// Mitsubishi GX Works2 project: Q03udv LG   PLC: Q03UDV
// ZONE 6 MOD 2021 06072021

PROGRAM MAIN
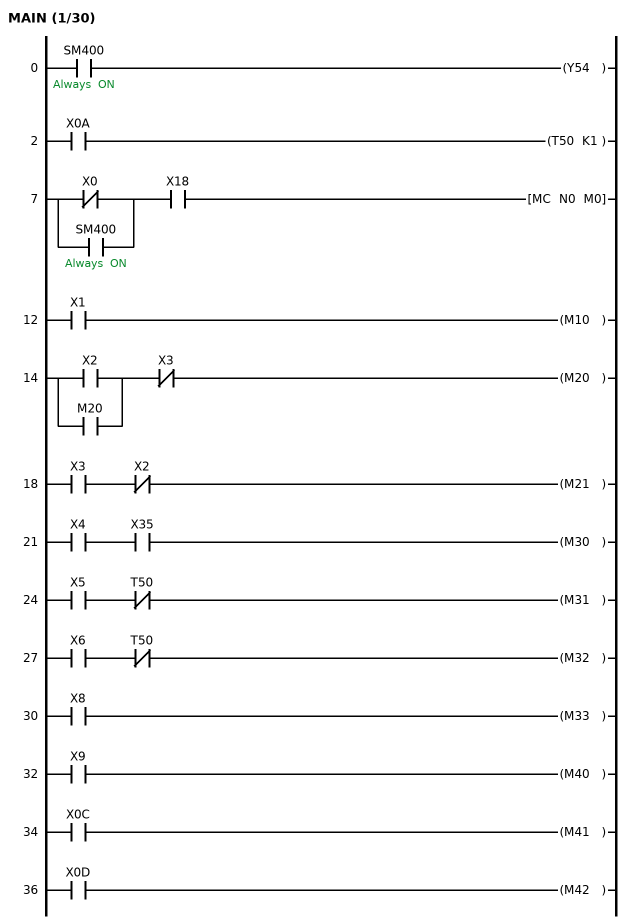
0     LD      SM400  ; Always  ON
      OUT     Y54
2     LD      X0A
      OUT     T50 K1
7     LDI     X0
      OR      SM400  ; Always  ON
      AND     X18
      MC      N0 M0
12    LD      X1
      OUT     M10
14    LD      X2
      OR      M20
      ANI     X3
      OUT     M20
18    LD      X3
      ANI     X2
      OUT     M21
21    LD      X4
      AND     X35
      OUT     M30
24    LD      X5
      ANI     T50
      OUT     M31
27    LD      X6
      ANI     T50
      OUT     M32
30    LD      X8
      OUT     M33
32    LD      X9
      OUT     M40
34    LD      X0C
      OUT     M41
36    LD      X0D
      OUT     M42
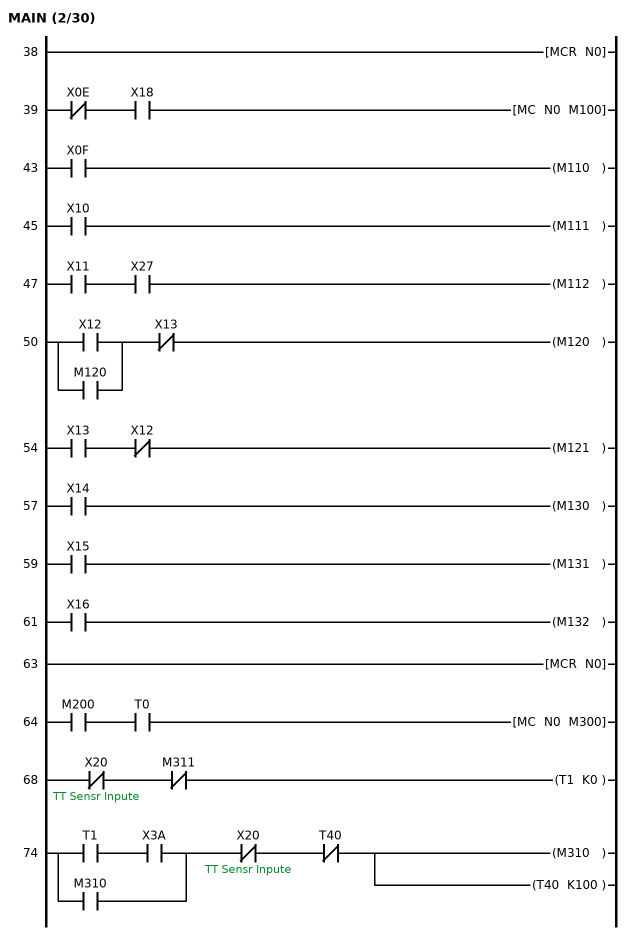
38    MCR     N0
39    LDI     X0E
      AND     X18
      MC      N0 M100
43    LD      X0F
      OUT     M110
45    LD      X10
      OUT     M111
47    LD      X11
      AND     X27
      OUT     M112
50    LD      X12
      OR      M120
      ANI     X13
      OUT     M120
54    LD      X13
      ANI     X12
      OUT     M121
57    LD      X14
      OUT     M130
59    LD      X15
      OUT     M131
61    LD      X16
      OUT     M132
63    MCR     N0
64    LD      M200
      AND     T0
      MC      N0 M300
68    LDI     X20  ; TT Sensr Inpute
      ANI     M311
      OUT     T1 K0
74    LD      T1
      AND     X3A
      OR      M310
      ANI     X20  ; TT Sensr Inpute
      ANI     T40
      OUT     M310
      OUT     T40 K100
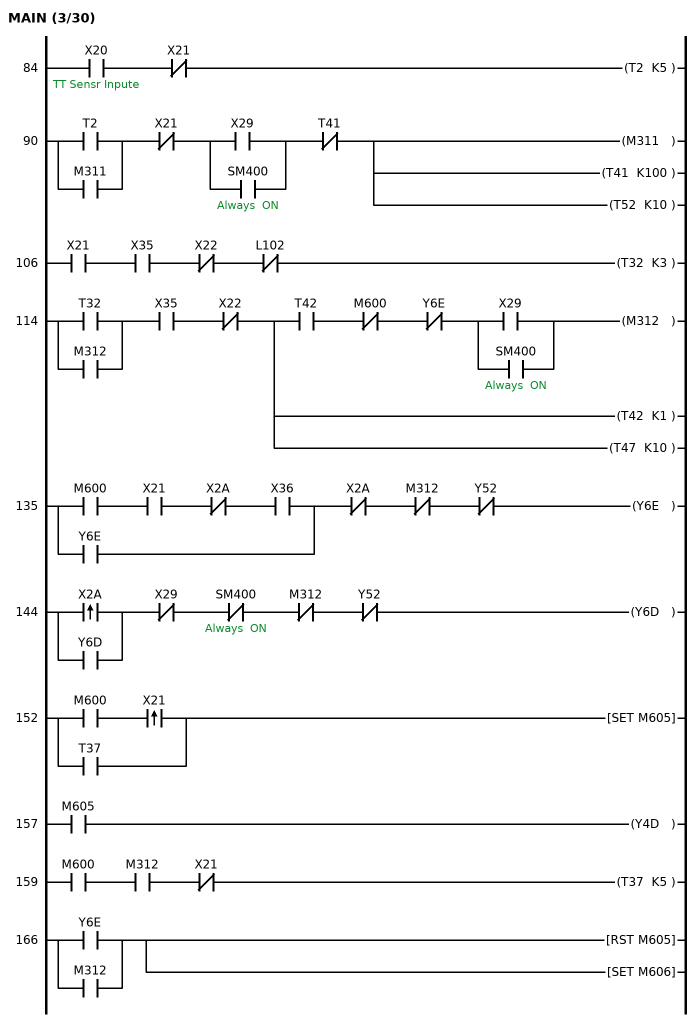
84    LD      X20  ; TT Sensr Inpute
      ANI     X21
      OUT     T2 K5
90    LD      T2
      OR      M311
      ANI     X21
      LD      X29
      OR      SM400  ; Always  ON
      ANB
      ANI     T41
      OUT     M311
      OUT     T41 K100
      OUT     T52 K10
106   LD      X21
      AND     X35
      ANI     X22
      ANI     L102
      OUT     T32 K3
114   LD      T32
      OR      M312
      AND     X35
      ANI     X22
      MPS
      AND     T42
      ANI     M600
      ANI     Y6E
      LD      X29
      OR      SM400  ; Always  ON
      ANB
      OUT     M312
      MPP
      OUT     T42 K1
      OUT     T47 K10
135   LD      M600
      AND     X21
      ANI     X2A
      AND     X36
      OR      Y6E
      ANI     X2A
      ANI     M312
      ANI     Y52
      OUT     Y6E
144   LDP     X2A
      OR      Y6D
      ANI     X29
      ANI     SM400  ; Always  ON
      ANI     M312
      ANI     Y52
      OUT     Y6D
152   LD      M600
      ANDP    X21
      OR      T37
      SET     M605
157   LD      M605
      OUT     Y4D
159   LD      M600
      AND     M312
      ANI     X21
      OUT     T37 K5
166   LD      Y6E
      OR      M312
      RST     M605
      SET     M606
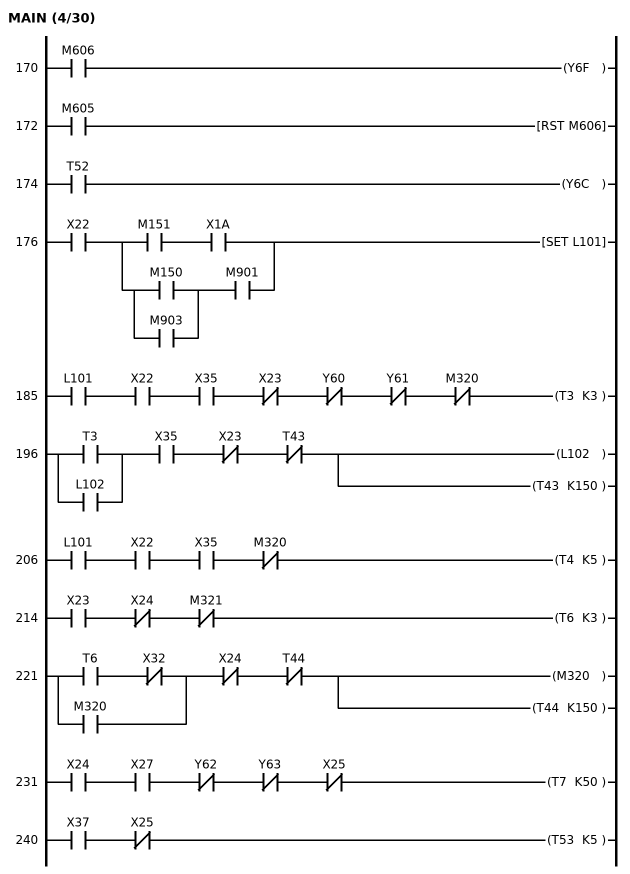
170   LD      M606
      OUT     Y6F
172   LD      M605
      RST     M606
174   LD      T52
      OUT     Y6C
176   LD      X22
      LD      M151
      AND     X1A
      LD      M150
      OR      M903
      AND     M901
      ORB
      ANB
      SET     L101
185   LD      L101
      AND     X22
      AND     X35
      ANI     X23
      ANI     Y60
      ANI     Y61
      ANI     M320
      OUT     T3 K3
196   LD      T3
      OR      L102
      AND     X35
      ANI     X23
      ANI     T43
      OUT     L102
      OUT     T43 K150
206   LD      L101
      AND     X22
      AND     X35
      ANI     M320
      OUT     T4 K5
214   LD      X23
      ANI     X24
      ANI     M321
      OUT     T6 K3
221   LD      T6
      ANI     X32
      OR      M320
      ANI     X24
      ANI     T44
      OUT     M320
      OUT     T44 K150
231   LD      X24
      AND     X27
      ANI     Y62
      ANI     Y63
      ANI     X25
      OUT     T7 K50
240   LD      X37
      ANI     X25
      OUT     T53 K5
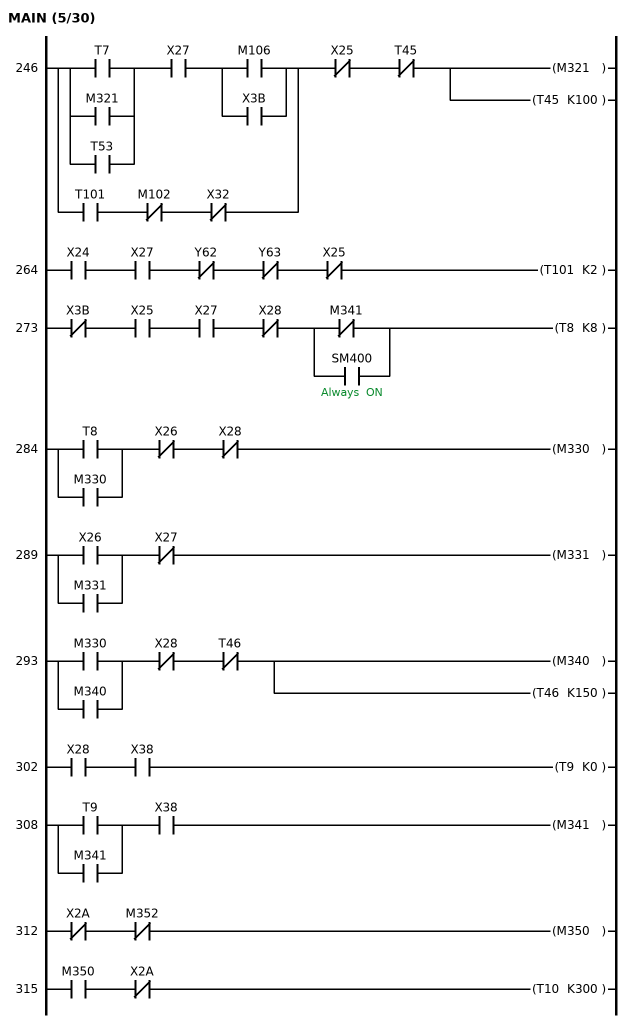
246   LD      T7
      OR      M321
      OR      T53
      AND     X27
      LD      M106
      OR      X3B
      ANB
      LD      T101
      ANI     M102
      ANI     X32
      ORB
      ANI     X25
      ANI     T45
      OUT     M321
      OUT     T45 K100
264   LD      X24
      AND     X27
      ANI     Y62
      ANI     Y63
      ANI     X25
      OUT     T101 K2
273   LDI     X3B
      AND     X25
      AND     X27
      ANI     X28
      LDI     M341
      OR      SM400  ; Always  ON
      ANB
      OUT     T8 K8
284   LD      T8
      OR      M330
      ANI     X26
      ANI     X28
      OUT     M330
289   LD      X26
      OR      M331
      ANI     X27
      OUT     M331
293   LD      M330
      OR      M340
      ANI     X28
      ANI     T46
      OUT     M340
      OUT     T46 K150
302   LD      X28
      AND     X38
      OUT     T9 K0
308   LD      T9
      OR      M341
      AND     X38
      OUT     M341
312   LDI     X2A
      ANI     M352
      OUT     M350
315   LD      M350
      ANI     X2A
      OUT     T10 K300
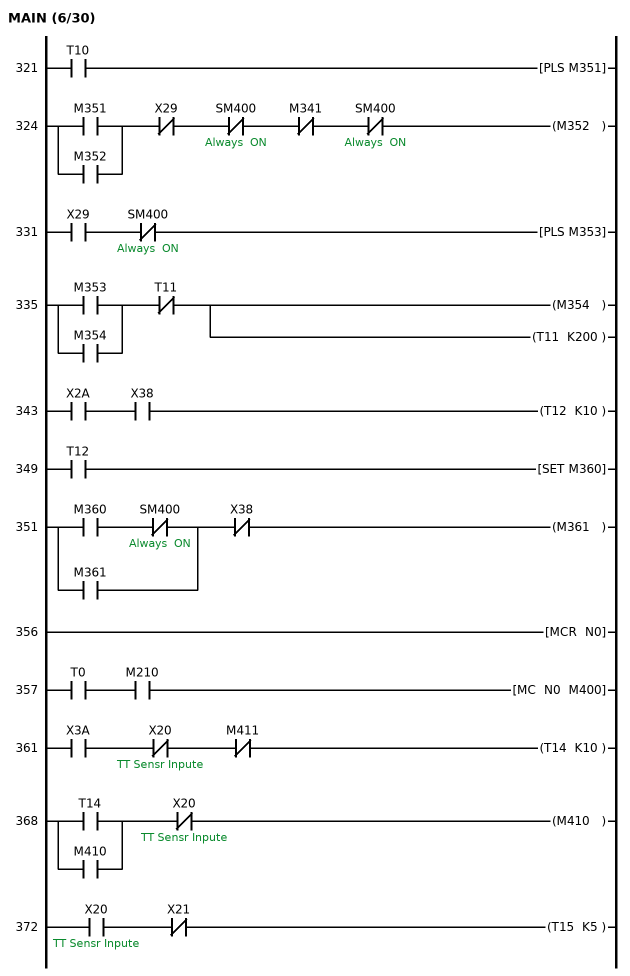
321   LD      T10
      PLS     M351
324   LD      M351
      OR      M352
      ANI     X29
      ANI     SM400  ; Always  ON
      ANI     M341
      ANI     SM400  ; Always  ON
      OUT     M352
331   LD      X29
      ANI     SM400  ; Always  ON
      PLS     M353
335   LD      M353
      OR      M354
      ANI     T11
      OUT     M354
      OUT     T11 K200
343   LD      X2A
      AND     X38
      OUT     T12 K10
349   LD      T12
      SET     M360
351   LD      M360
      ANI     SM400  ; Always  ON
      OR      M361
      ANI     X38
      OUT     M361
356   MCR     N0
357   LD      T0
      AND     M210
      MC      N0 M400
361   LD      X3A
      ANI     X20  ; TT Sensr Inpute
      ANI     M411
      OUT     T14 K10
368   LD      T14
      OR      M410
      ANI     X20  ; TT Sensr Inpute
      OUT     M410
372   LD      X20  ; TT Sensr Inpute
      ANI     X21
      OUT     T15 K5
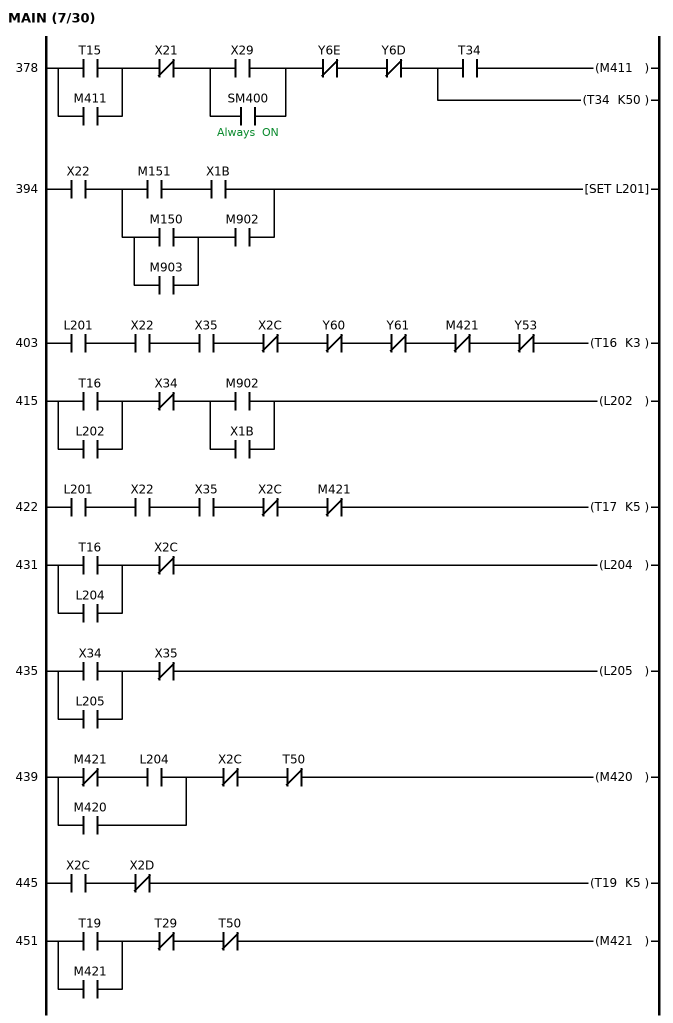
378   LD      T15
      OR      M411
      ANI     X21
      LD      X29
      OR      SM400  ; Always  ON
      ANB
      ANI     Y6E
      ANI     Y6D
      MPS
      AND     T34
      OUT     M411
      MPP
      OUT     T34 K50
394   LD      X22
      LD      M151
      AND     X1B
      LD      M150
      OR      M903
      AND     M902
      ORB
      ANB
      SET     L201
403   LD      L201
      AND     X22
      AND     X35
      ANI     X2C
      ANI     Y60
      ANI     Y61
      ANI     M421
      ANI     Y53
      OUT     T16 K3
415   LD      T16
      OR      L202
      ANI     X34
      LD      M902
      OR      X1B
      ANB
      OUT     L202
422   LD      L201
      AND     X22
      AND     X35
      ANI     X2C
      ANI     M421
      OUT     T17 K5
431   LD      T16
      OR      L204
      ANI     X2C
      OUT     L204
435   LD      X34
      OR      L205
      ANI     X35
      OUT     L205
439   LDI     M421
      AND     L204
      OR      M420
      ANI     X2C
      ANI     T50
      OUT     M420
445   LD      X2C
      ANI     X2D
      OUT     T19 K5
451   LD      T19
      OR      M421
      ANI     T29
      ANI     T50
      OUT     M421
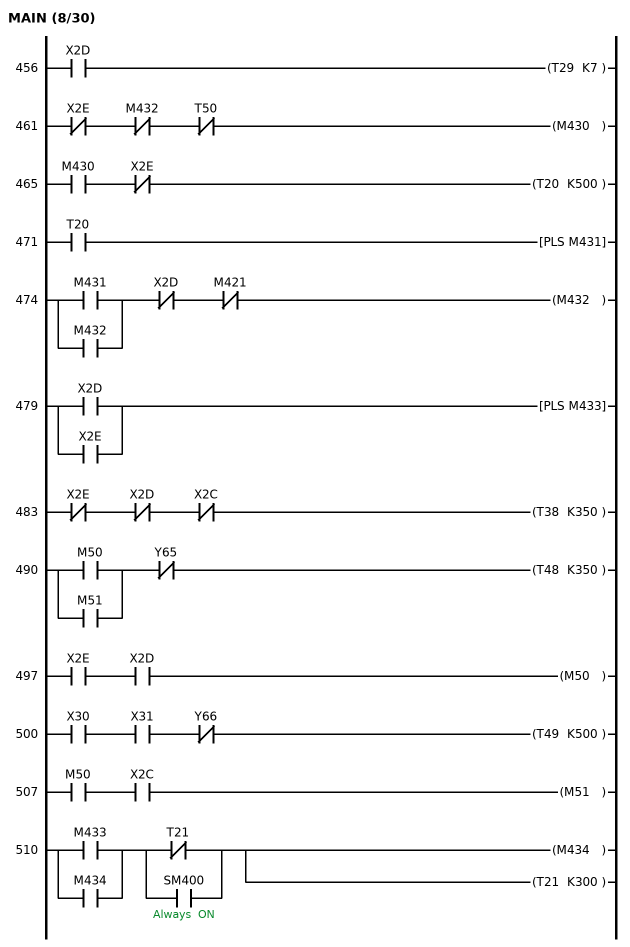
456   LD      X2D
      OUT     T29 K7
461   LDI     X2E
      ANI     M432
      ANI     T50
      OUT     M430
465   LD      M430
      ANI     X2E
      OUT     T20 K500
471   LD      T20
      PLS     M431
474   LD      M431
      OR      M432
      ANI     X2D
      ANI     M421
      OUT     M432
479   LD      X2D
      OR      X2E
      PLS     M433
483   LDI     X2E
      ANI     X2D
      ANI     X2C
      OUT     T38 K350
490   LD      M50
      OR      M51
      ANI     Y65
      OUT     T48 K350
497   LD      X2E
      AND     X2D
      OUT     M50
500   LD      X30
      AND     X31
      ANI     Y66
      OUT     T49 K500
507   LD      M50
      AND     X2C
      OUT     M51
510   LD      M433
      OR      M434
      LDI     T21
      OR      SM400  ; Always  ON
      ANB
      OUT     M434
      OUT     T21 K300
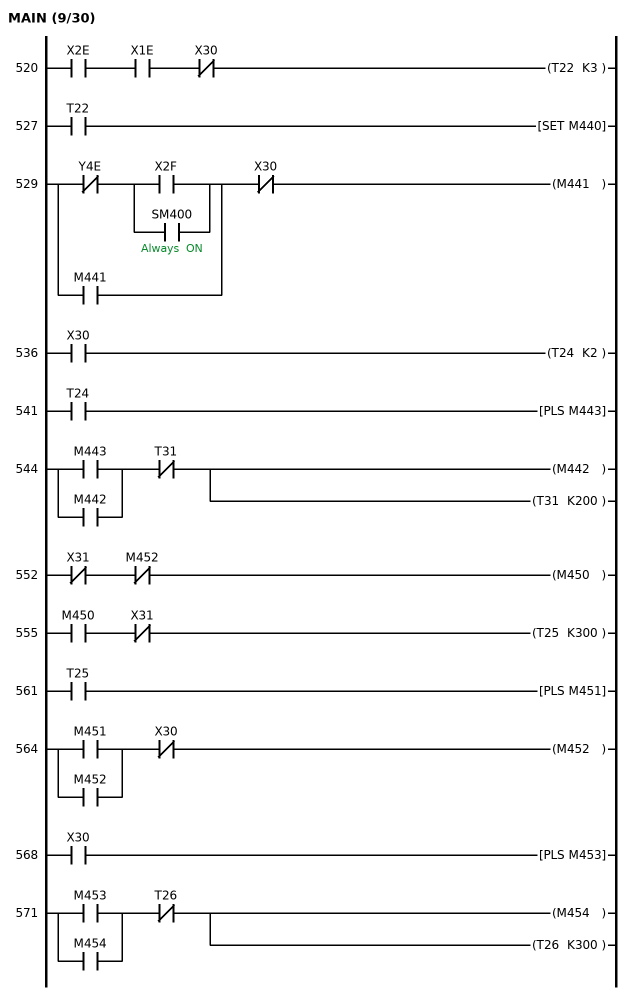
520   LD      X2E
      AND     X1E
      ANI     X30
      OUT     T22 K3
527   LD      T22
      SET     M440
529   LDI     Y4E
      LD      X2F
      OR      SM400  ; Always  ON
      ANB
      OR      M441
      ANI     X30
      OUT     M441
536   LD      X30
      OUT     T24 K2
541   LD      T24
      PLS     M443
544   LD      M443
      OR      M442
      ANI     T31
      OUT     M442
      OUT     T31 K200
552   LDI     X31
      ANI     M452
      OUT     M450
555   LD      M450
      ANI     X31
      OUT     T25 K300
561   LD      T25
      PLS     M451
564   LD      M451
      OR      M452
      ANI     X30
      OUT     M452
568   LD      X30
      PLS     M453
571   LD      M453
      OR      M454
      ANI     T26
      OUT     M454
      OUT     T26 K300
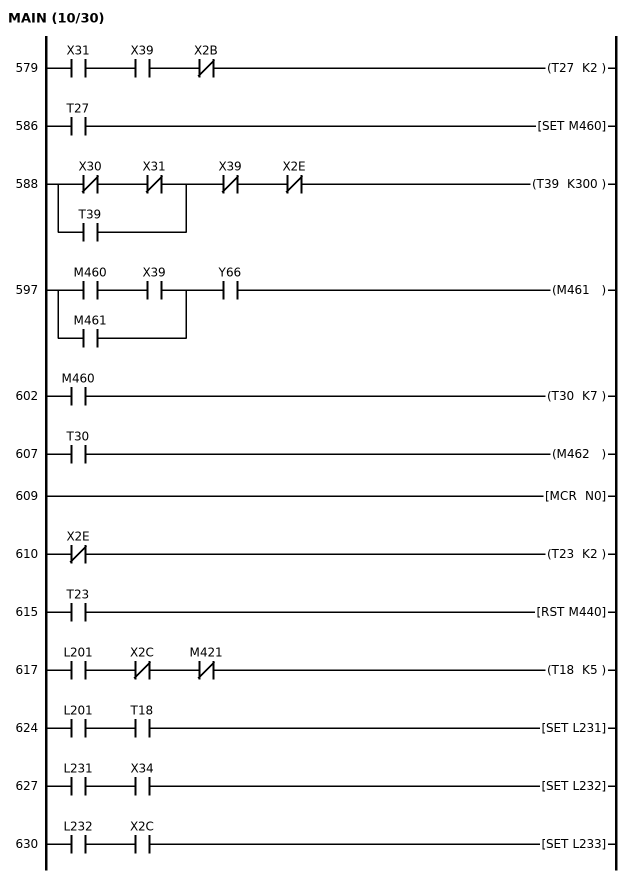
579   LD      X31
      AND     X39
      ANI     X2B
      OUT     T27 K2
586   LD      T27
      SET     M460
588   LDI     X30
      ANI     X31
      OR      T39
      ANI     X39
      ANI     X2E
      OUT     T39 K300
597   LD      M460
      AND     X39
      OR      M461
      AND     Y66
      OUT     M461
602   LD      M460
      OUT     T30 K7
607   LD      T30
      OUT     M462
609   MCR     N0
610   LDI     X2E
      OUT     T23 K2
615   LD      T23
      RST     M440
617   LD      L201
      ANI     X2C
      ANI     M421
      OUT     T18 K5
624   LD      L201
      AND     T18
      SET     L231
627   LD      L231
      AND     X34
      SET     L232
630   LD      L232
      AND     X2C
      SET     L233
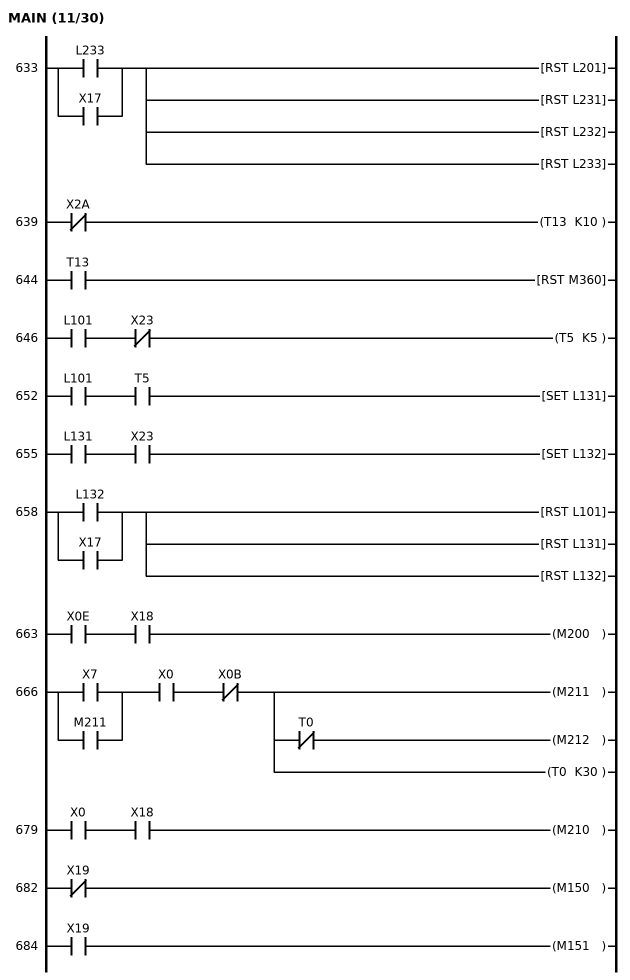
633   LD      L233
      OR      X17
      RST     L201
      RST     L231
      RST     L232
      RST     L233
639   LDI     X2A
      OUT     T13 K10
644   LD      T13
      RST     M360
646   LD      L101
      ANI     X23
      OUT     T5 K5
652   LD      L101
      AND     T5
      SET     L131
655   LD      L131
      AND     X23
      SET     L132
658   LD      L132
      OR      X17
      RST     L101
      RST     L131
      RST     L132
663   LD      X0E
      AND     X18
      OUT     M200
666   LD      X7
      OR      M211
      AND     X0
      ANI     X0B
      OUT     M211
      MPS
      ANI     T0
      OUT     M212
      MPP
      OUT     T0 K30
679   LD      X0
      AND     X18
      OUT     M210
682   LDI     X19
      OUT     M150
684   LD      X19
      OUT     M151
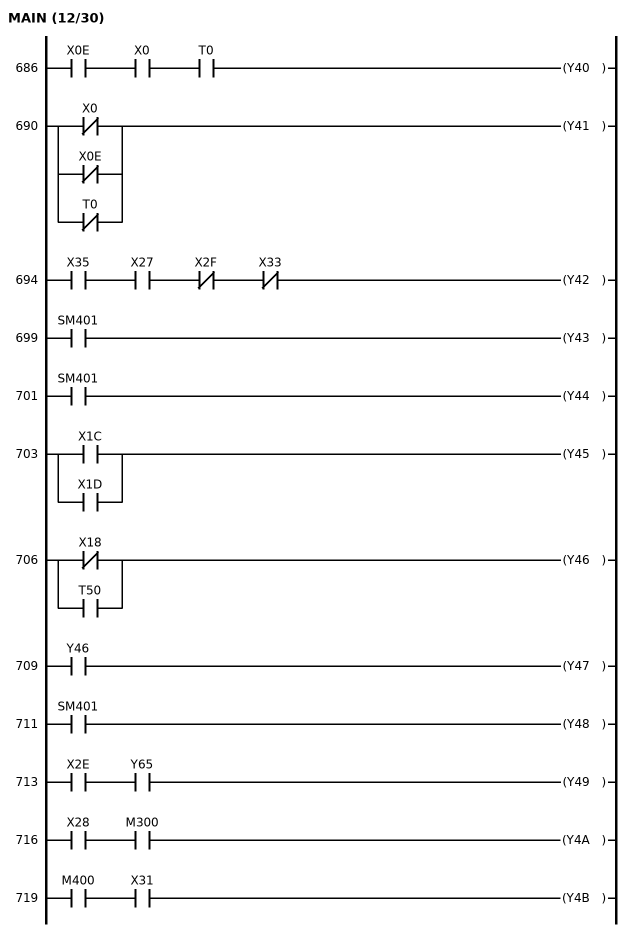
686   LD      X0E
      AND     X0
      AND     T0
      OUT     Y40
690   LDI     X0
      ORI     X0E
      ORI     T0
      OUT     Y41
694   LD      X35
      AND     X27
      ANI     X2F
      ANI     X33
      OUT     Y42
699   LD      SM401
      OUT     Y43
701   LD      SM401
      OUT     Y44
703   LD      X1C
      OR      X1D
      OUT     Y45
706   LDI     X18
      OR      T50
      OUT     Y46
709   LD      Y46
      OUT     Y47
711   LD      SM401
      OUT     Y48
713   LD      X2E
      AND     Y65
      OUT     Y49
716   LD      X28
      AND     M300
      OUT     Y4A
719   LD      M400
      AND     X31
      OUT     Y4B
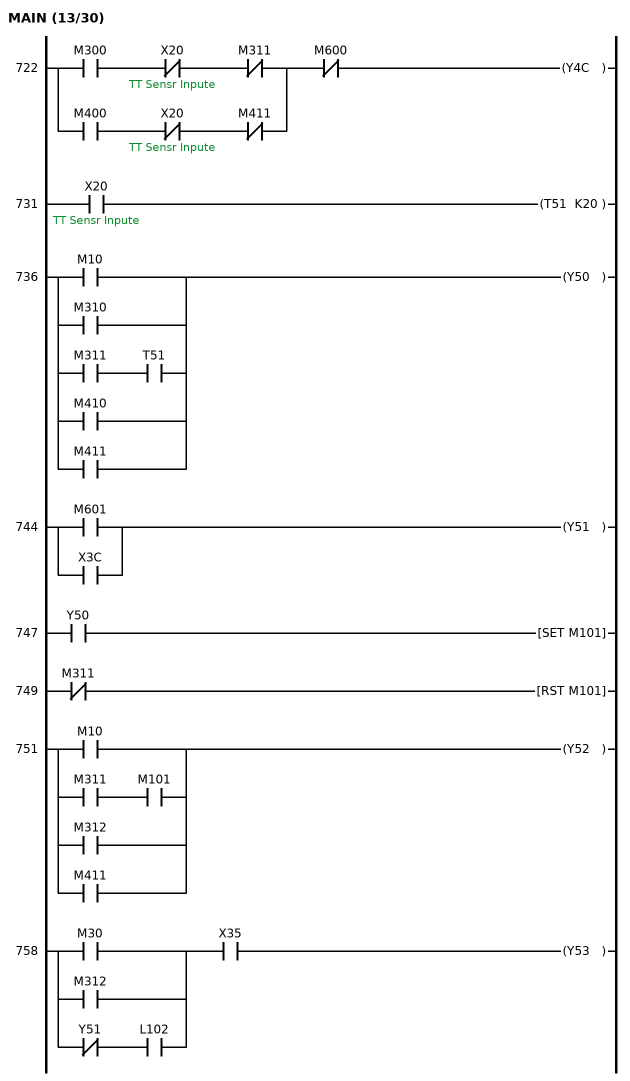
722   LD      M300
      ANI     X20  ; TT Sensr Inpute
      ANI     M311
      LD      M400
      ANI     X20  ; TT Sensr Inpute
      ANI     M411
      ORB
      ANI     M600
      OUT     Y4C
731   LD      X20  ; TT Sensr Inpute
      OUT     T51 K20
736   LD      M10
      OR      M310
      LD      M311
      AND     T51
      ORB
      OR      M410
      OR      M411
      OUT     Y50
744   LD      M601
      OR      X3C
      OUT     Y51
747   LD      Y50
      SET     M101
749   LDI     M311
      RST     M101
751   LD      M10
      LD      M311
      AND     M101
      ORB
      OR      M312
      OR      M411
      OUT     Y52
758   LD      M30
      OR      M312
      LDI     Y51
      AND     L102
      ORB
      AND     X35
      OUT     Y53
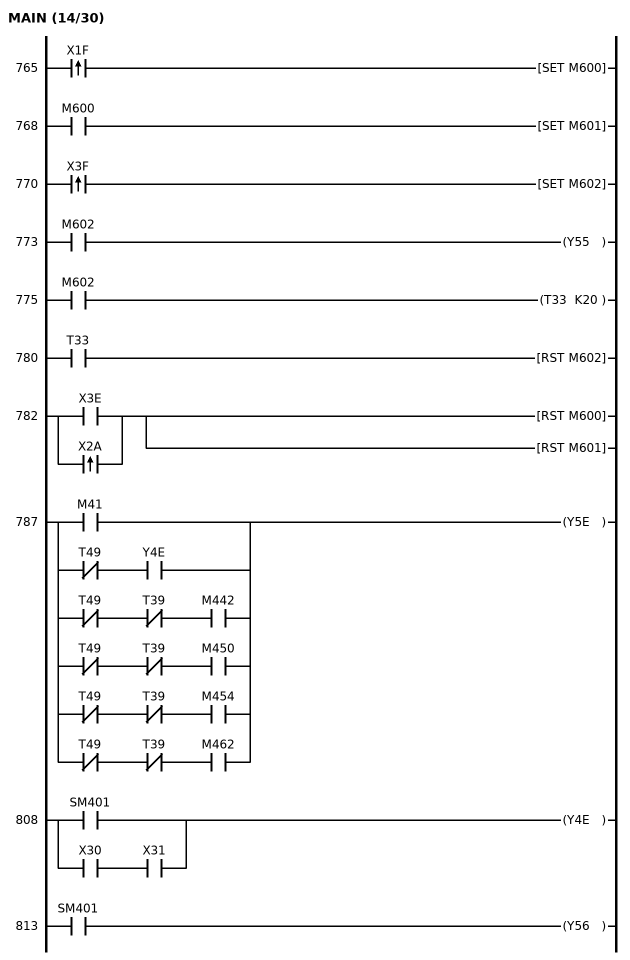
765   LDP     X1F
      SET     M600
768   LD      M600
      SET     M601
770   LDP     X3F
      SET     M602
773   LD      M602
      OUT     Y55
775   LD      M602
      OUT     T33 K20
780   LD      T33
      RST     M602
782   LD      X3E
      ORP     X2A
      RST     M600
      RST     M601
787   LD      M41
      LDI     T49
      AND     Y4E
      ORB
      LDI     T49
      ANI     T39
      AND     M442
      ORB
      LDI     T49
      ANI     T39
      AND     M450
      ORB
      LDI     T49
      ANI     T39
      AND     M454
      ORB
      LDI     T49
      ANI     T39
      AND     M462
      ORB
      OUT     Y5E
808   LD      SM401
      LD      X30
      AND     X31
      ORB
      OUT     Y4E
813   LD      SM401
      OUT     Y56
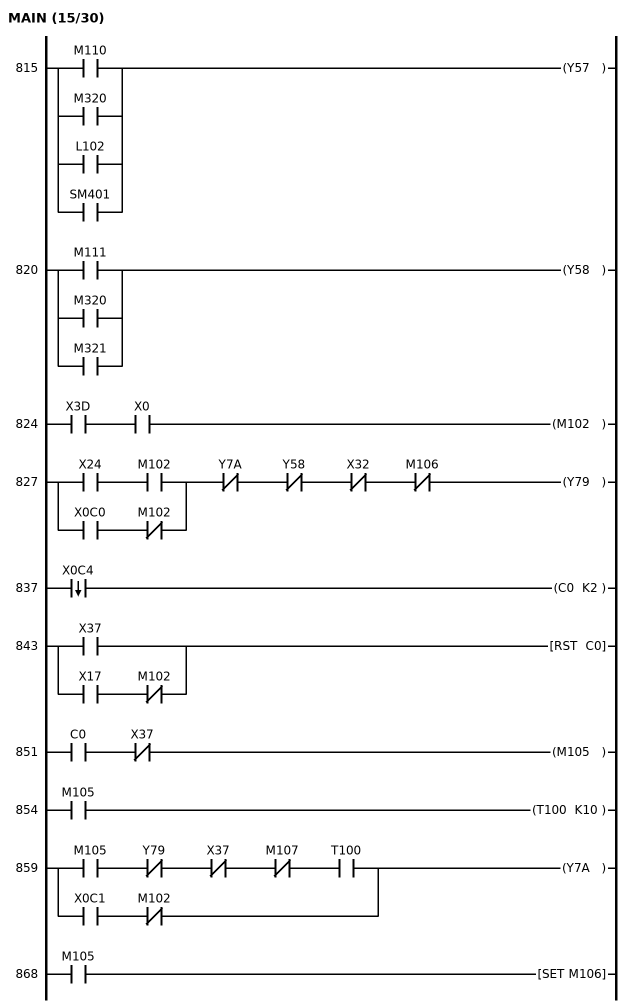
815   LD      M110
      OR      M320
      OR      L102
      OR      SM401
      OUT     Y57
820   LD      M111
      OR      M320
      OR      M321
      OUT     Y58
824   LD      X3D
      AND     X0
      OUT     M102
827   LD      X24
      AND     M102
      LD      X0C0
      ANI     M102
      ORB
      ANI     Y7A
      ANI     Y58
      ANI     X32
      ANI     M106
      OUT     Y79
837   LDF     X0C4
      OUT     C0 K2
843   LD      X37
      LD      X17
      ANI     M102
      ORB
      RST     C0
851   LD      C0
      ANI     X37
      OUT     M105
854   LD      M105
      OUT     T100 K10
859   LD      M105
      ANI     Y79
      ANI     X37
      ANI     M107
      AND     T100
      LD      X0C1
      ANI     M102
      ORB
      OUT     Y7A
868   LD      M105
      SET     M106
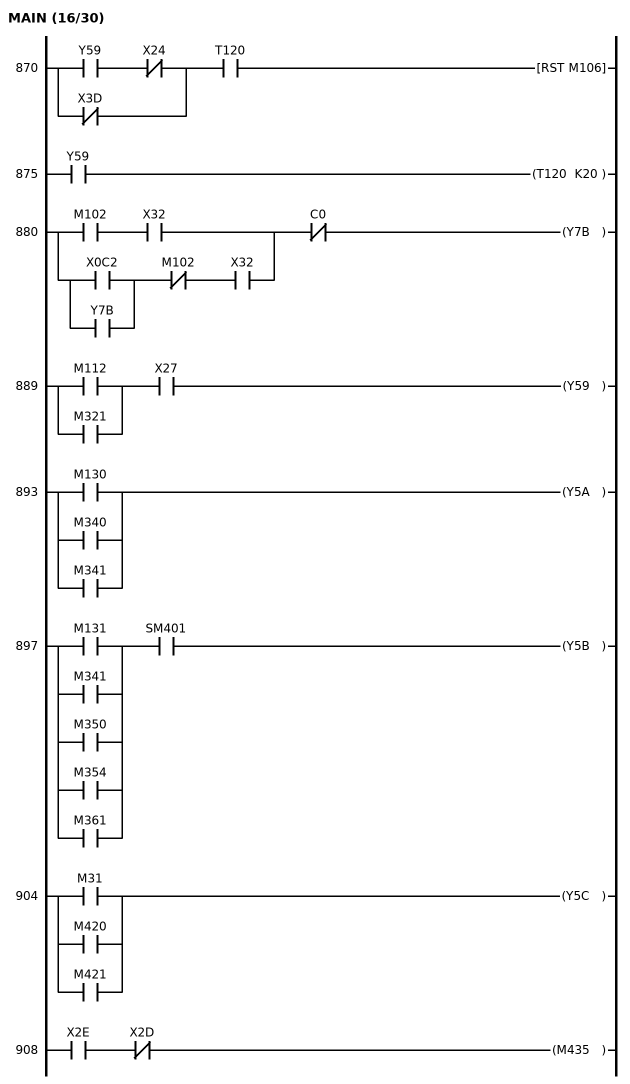
870   LD      Y59
      ANI     X24
      ORI     X3D
      AND     T120
      RST     M106
875   LD      Y59
      OUT     T120 K20
880   LD      M102
      AND     X32
      LD      X0C2
      OR      Y7B
      ANI     M102
      AND     X32
      ORB
      ANI     C0
      OUT     Y7B
889   LD      M112
      OR      M321
      AND     X27
      OUT     Y59
893   LD      M130
      OR      M340
      OR      M341
      OUT     Y5A
897   LD      M131
      OR      M341
      OR      M350
      OR      M354
      OR      M361
      AND     SM401
      OUT     Y5B
904   LD      M31
      OR      M420
      OR      M421
      OUT     Y5C
908   LD      X2E
      ANI     X2D
      OUT     M435
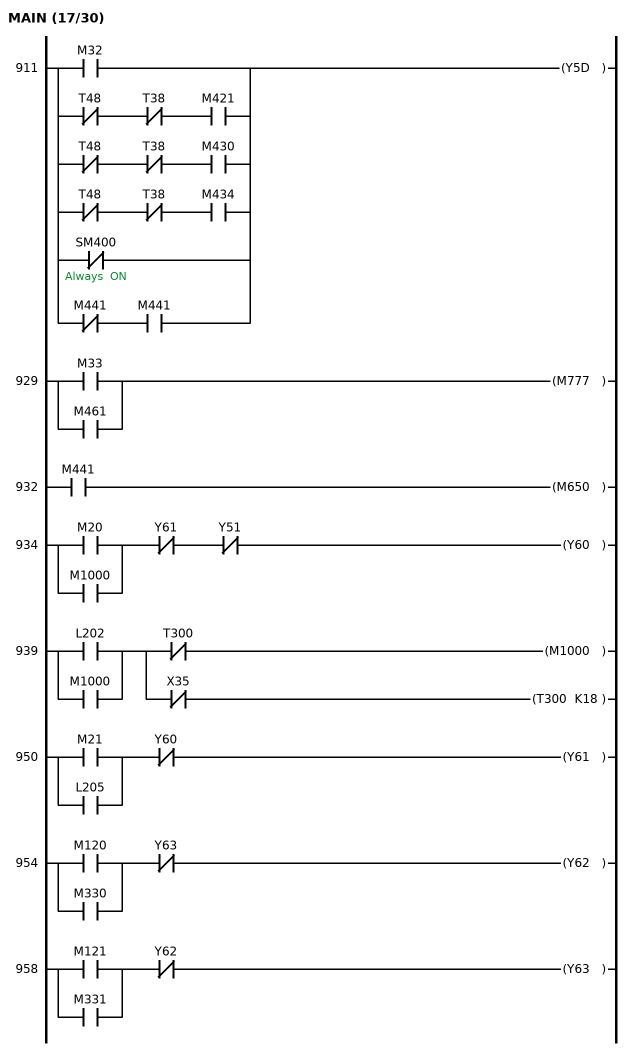
911   LD      M32
      LDI     T48
      ANI     T38
      AND     M421
      ORB
      LDI     T48
      ANI     T38
      AND     M430
      ORB
      LDI     T48
      ANI     T38
      AND     M434
      ORB
      ORI     SM400  ; Always  ON
      LDI     M441
      AND     M441
      ORB
      OUT     Y5D
929   LD      M33
      OR      M461
      OUT     M777
932   LD      M441
      OUT     M650
934   LD      M20
      OR      M1000
      ANI     Y61
      ANI     Y51
      OUT     Y60
939   LD      L202
      OR      M1000
      MPS
      ANI     T300
      OUT     M1000
      MPP
      ANI     X35
      OUT     T300 K18
950   LD      M21
      OR      L205
      ANI     Y60
      OUT     Y61
954   LD      M120
      OR      M330
      ANI     Y63
      OUT     Y62
958   LD      M121
      OR      M331
      ANI     Y62
      OUT     Y63
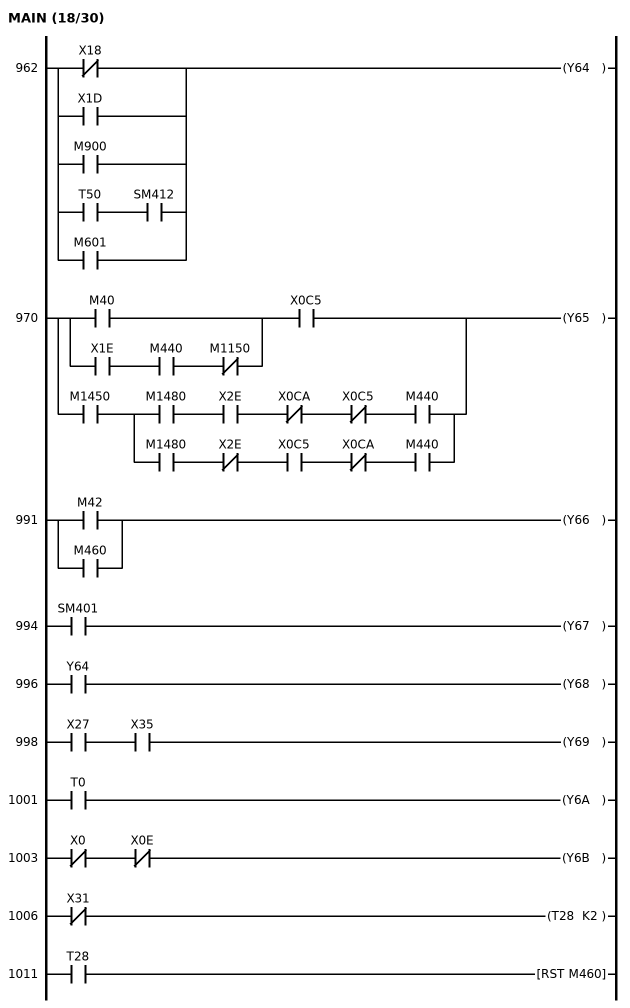
962   LDI     X18
      OR      X1D
      OR      M900
      LD      T50
      AND     SM412
      ORB
      OR      M601
      OUT     Y64
970   LD      M40
      LD      X1E
      AND     M440
      ANI     M1150
      ORB
      AND     X0C5
      LD      M1450
      LD      M1480
      AND     X2E
      ANI     X0CA
      ANI     X0C5
      AND     M440
      LD      M1480
      ANI     X2E
      AND     X0C5
      ANI     X0CA
      AND     M440
      ORB
      ANB
      ORB
      OUT     Y65
991   LD      M42
      OR      M460
      OUT     Y66
994   LD      SM401
      OUT     Y67
996   LD      Y64
      OUT     Y68
998   LD      X27
      AND     X35
      OUT     Y69
1001  LD      T0
      OUT     Y6A
1003  LDI     X0
      ANI     X0E
      OUT     Y6B
1006  LDI     X31
      OUT     T28 K2
1011  LD      T28
      RST     M460
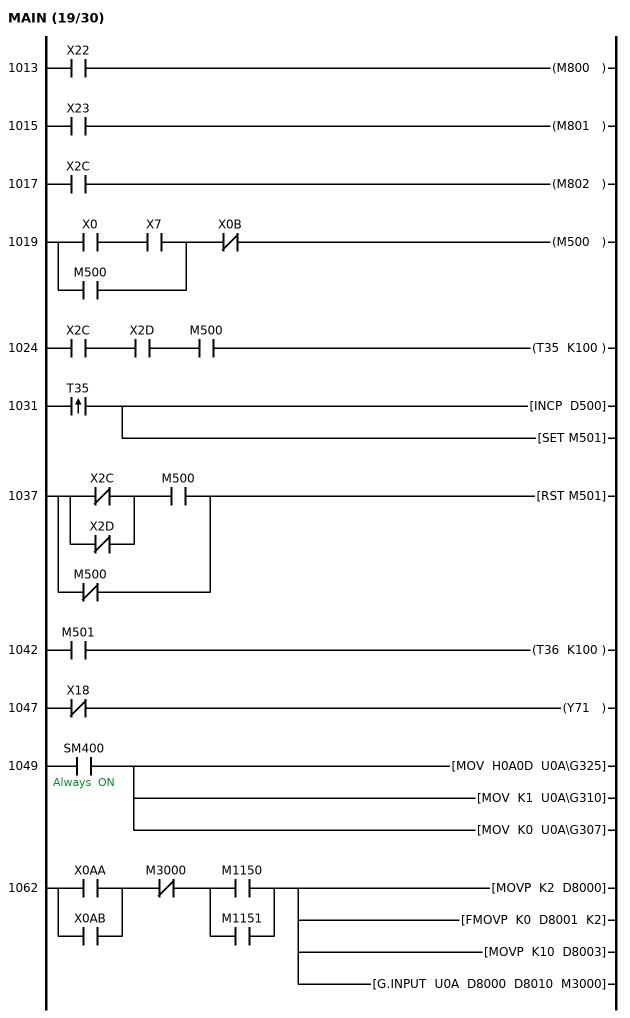
1013  LD      X22
      OUT     M800
1015  LD      X23
      OUT     M801
1017  LD      X2C
      OUT     M802
1019  LD      X0
      AND     X7
      OR      M500
      ANI     X0B
      OUT     M500
1024  LD      X2C
      AND     X2D
      AND     M500
      OUT     T35 K100
1031  LDP     T35
      INCP    D500
      SET     M501
1037  LDI     X2C
      ORI     X2D
      AND     M500
      ORI     M500
      RST     M501
1042  LD      M501
      OUT     T36 K100
1047  LDI     X18
      OUT     Y71
1049  LD      SM400  ; Always  ON
      MOV     H0A0D U0A\G325
      MOV     K1 U0A\G310
      MOV     K0 U0A\G307
1062  LD      X0AA
      OR      X0AB
      ANI     M3000
      LD      M1150
      OR      M1151
      ANB
      MOVP    K2 D8000
      FMOVP   K0 D8001 K2
      MOVP    K10 D8003
      G.INPUT U0A D8000 D8010 M3000
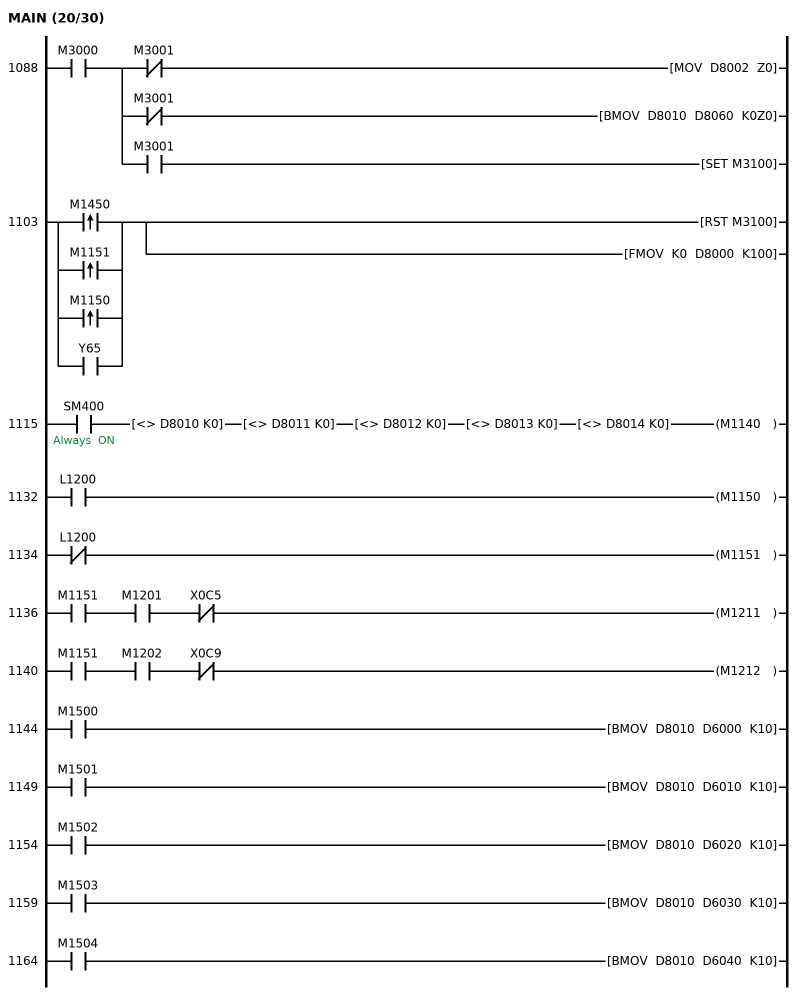
1088  LD      M3000
      MPS
      ANI     M3001
      MOV     D8002 Z0
      MRD
      ANI     M3001
      BMOV    D8010 D8060 K0Z0
      MPP
      AND     M3001
      SET     M3100
1103  LDP     M1450
      ORP     M1151
      ORP     M1150
      OR      Y65
      RST     M3100
      FMOV    K0 D8000 K100
1115  LD      SM400  ; Always  ON
      AND<>   D8010 K0
      AND<>   D8011 K0
      AND<>   D8012 K0
      AND<>   D8013 K0
      AND<>   D8014 K0
      OUT     M1140
1132  LD      L1200
      OUT     M1150
1134  LDI     L1200
      OUT     M1151
1136  LD      M1151
      AND     M1201
      ANI     X0C5
      OUT     M1211
1140  LD      M1151
      AND     M1202
      ANI     X0C9
      OUT     M1212
1144  LD      M1500
      BMOV    D8010 D6000 K10
1149  LD      M1501
      BMOV    D8010 D6010 K10
1154  LD      M1502
      BMOV    D8010 D6020 K10
1159  LD      M1503
      BMOV    D8010 D6030 K10
1164  LD      M1504
      BMOV    D8010 D6040 K10
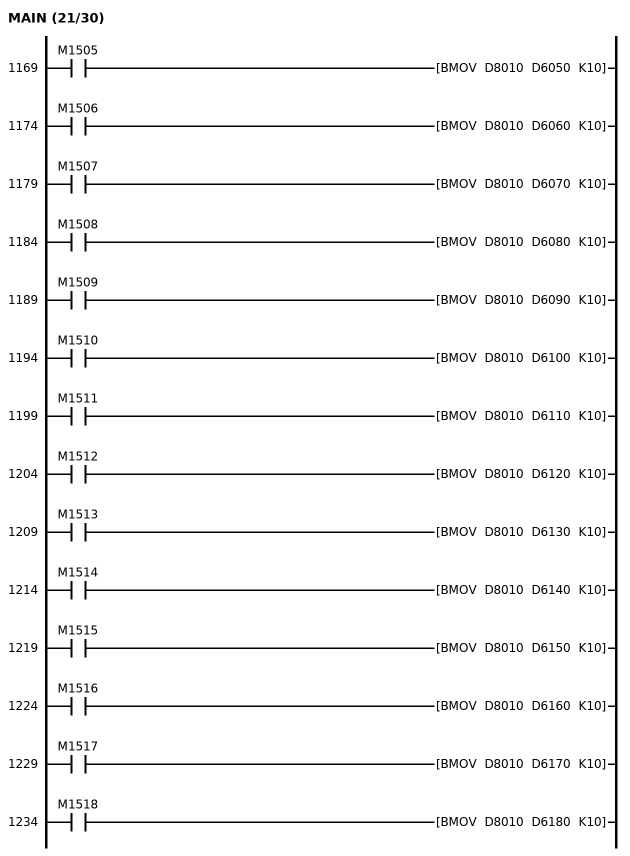
1169  LD      M1505
      BMOV    D8010 D6050 K10
1174  LD      M1506
      BMOV    D8010 D6060 K10
1179  LD      M1507
      BMOV    D8010 D6070 K10
1184  LD      M1508
      BMOV    D8010 D6080 K10
1189  LD      M1509
      BMOV    D8010 D6090 K10
1194  LD      M1510
      BMOV    D8010 D6100 K10
1199  LD      M1511
      BMOV    D8010 D6110 K10
1204  LD      M1512
      BMOV    D8010 D6120 K10
1209  LD      M1513
      BMOV    D8010 D6130 K10
1214  LD      M1514
      BMOV    D8010 D6140 K10
1219  LD      M1515
      BMOV    D8010 D6150 K10
1224  LD      M1516
      BMOV    D8010 D6160 K10
1229  LD      M1517
      BMOV    D8010 D6170 K10
1234  LD      M1518
      BMOV    D8010 D6180 K10
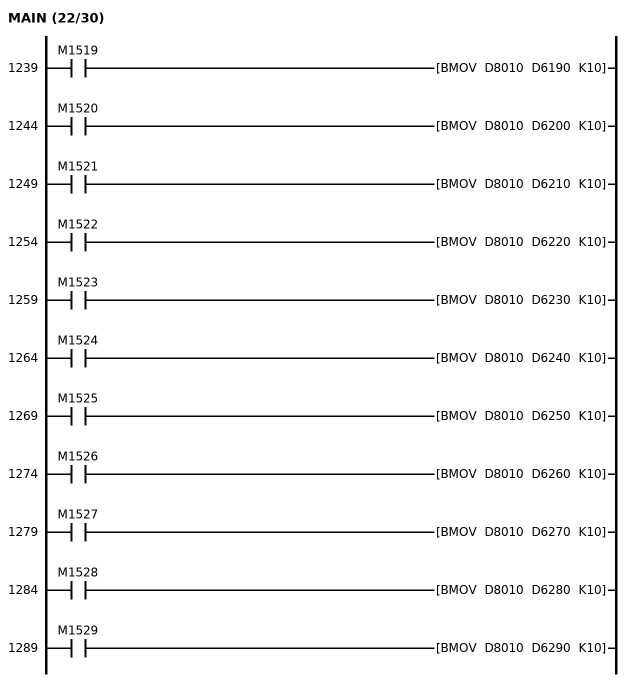
1239  LD      M1519
      BMOV    D8010 D6190 K10
1244  LD      M1520
      BMOV    D8010 D6200 K10
1249  LD      M1521
      BMOV    D8010 D6210 K10
1254  LD      M1522
      BMOV    D8010 D6220 K10
1259  LD      M1523
      BMOV    D8010 D6230 K10
1264  LD      M1524
      BMOV    D8010 D6240 K10
1269  LD      M1525
      BMOV    D8010 D6250 K10
1274  LD      M1526
      BMOV    D8010 D6260 K10
1279  LD      M1527
      BMOV    D8010 D6270 K10
1284  LD      M1528
      BMOV    D8010 D6280 K10
1289  LD      M1529
      BMOV    D8010 D6290 K10
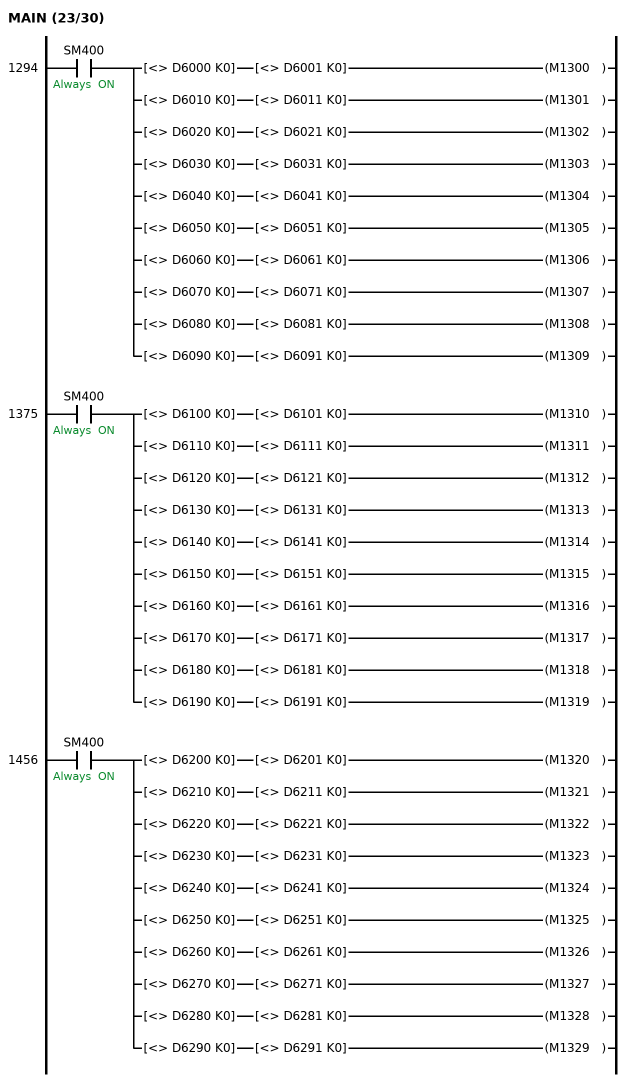
1294  LD      SM400  ; Always  ON
      MPS
      AND<>   D6000 K0
      AND<>   D6001 K0
      OUT     M1300
      MRD
      AND<>   D6010 K0
      AND<>   D6011 K0
      OUT     M1301
      MRD
      AND<>   D6020 K0
      AND<>   D6021 K0
      OUT     M1302
      MRD
      AND<>   D6030 K0
      AND<>   D6031 K0
      OUT     M1303
      MRD
      AND<>   D6040 K0
      AND<>   D6041 K0
      OUT     M1304
      MRD
      AND<>   D6050 K0
      AND<>   D6051 K0
      OUT     M1305
      MRD
      AND<>   D6060 K0
      AND<>   D6061 K0
      OUT     M1306
      MRD
      AND<>   D6070 K0
      AND<>   D6071 K0
      OUT     M1307
      MRD
      AND<>   D6080 K0
      AND<>   D6081 K0
      OUT     M1308
      MPP
      AND<>   D6090 K0
      AND<>   D6091 K0
      OUT     M1309
1375  LD      SM400  ; Always  ON
      MPS
      AND<>   D6100 K0
      AND<>   D6101 K0
      OUT     M1310
      MRD
      AND<>   D6110 K0
      AND<>   D6111 K0
      OUT     M1311
      MRD
      AND<>   D6120 K0
      AND<>   D6121 K0
      OUT     M1312
      MRD
      AND<>   D6130 K0
      AND<>   D6131 K0
      OUT     M1313
      MRD
      AND<>   D6140 K0
      AND<>   D6141 K0
      OUT     M1314
      MRD
      AND<>   D6150 K0
      AND<>   D6151 K0
      OUT     M1315
      MRD
      AND<>   D6160 K0
      AND<>   D6161 K0
      OUT     M1316
      MRD
      AND<>   D6170 K0
      AND<>   D6171 K0
      OUT     M1317
      MRD
      AND<>   D6180 K0
      AND<>   D6181 K0
      OUT     M1318
      MPP
      AND<>   D6190 K0
      AND<>   D6191 K0
      OUT     M1319
1456  LD      SM400  ; Always  ON
      MPS
      AND<>   D6200 K0
      AND<>   D6201 K0
      OUT     M1320
      MRD
      AND<>   D6210 K0
      AND<>   D6211 K0
      OUT     M1321
      MRD
      AND<>   D6220 K0
      AND<>   D6221 K0
      OUT     M1322
      MRD
      AND<>   D6230 K0
      AND<>   D6231 K0
      OUT     M1323
      MRD
      AND<>   D6240 K0
      AND<>   D6241 K0
      OUT     M1324
      MRD
      AND<>   D6250 K0
      AND<>   D6251 K0
      OUT     M1325
      MRD
      AND<>   D6260 K0
      AND<>   D6261 K0
      OUT     M1326
      MRD
      AND<>   D6270 K0
      AND<>   D6271 K0
      OUT     M1327
      MRD
      AND<>   D6280 K0
      AND<>   D6281 K0
      OUT     M1328
      MPP
      AND<>   D6290 K0
      AND<>   D6291 K0
      OUT     M1329
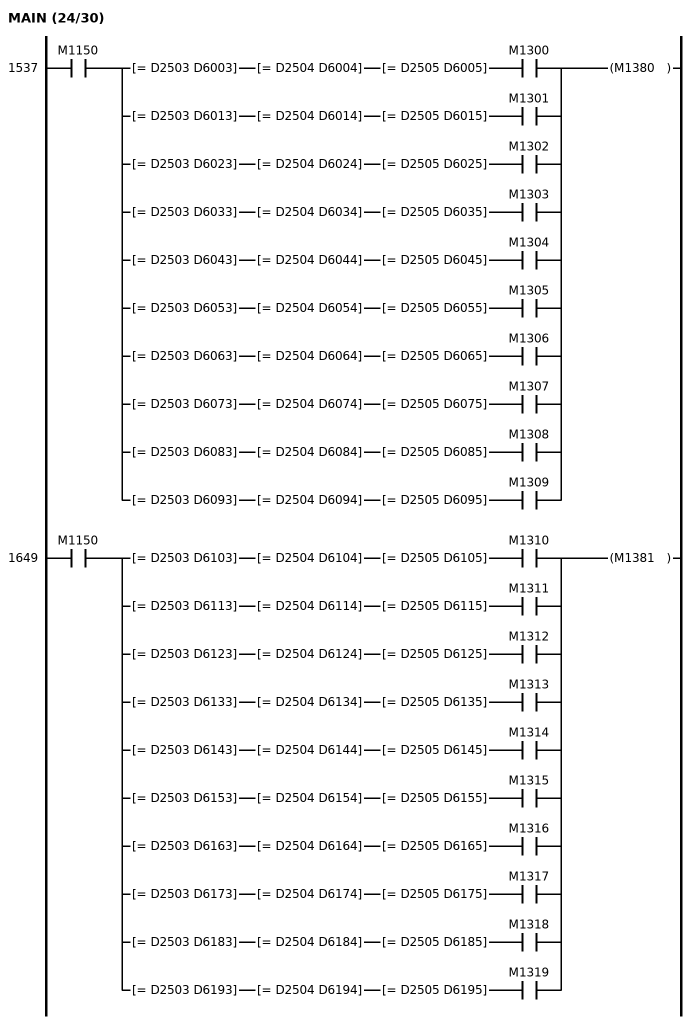
1537  LD      M1150
      LD=     D2503 D6003
      AND=    D2504 D6004
      AND=    D2505 D6005
      AND     M1300
      LD=     D2503 D6013
      AND=    D2504 D6014
      AND=    D2505 D6015
      AND     M1301
      ORB
      LD=     D2503 D6023
      AND=    D2504 D6024
      AND=    D2505 D6025
      AND     M1302
      ORB
      LD=     D2503 D6033
      AND=    D2504 D6034
      AND=    D2505 D6035
      AND     M1303
      ORB
      LD=     D2503 D6043
      AND=    D2504 D6044
      AND=    D2505 D6045
      AND     M1304
      ORB
      LD=     D2503 D6053
      AND=    D2504 D6054
      AND=    D2505 D6055
      AND     M1305
      ORB
      LD=     D2503 D6063
      AND=    D2504 D6064
      AND=    D2505 D6065
      AND     M1306
      ORB
      LD=     D2503 D6073
      AND=    D2504 D6074
      AND=    D2505 D6075
      AND     M1307
      ORB
      LD=     D2503 D6083
      AND=    D2504 D6084
      AND=    D2505 D6085
      AND     M1308
      ORB
      LD=     D2503 D6093
      AND=    D2504 D6094
      AND=    D2505 D6095
      AND     M1309
      ORB
      ANB
      OUT     M1380
1649  LD      M1150
      LD=     D2503 D6103
      AND=    D2504 D6104
      AND=    D2505 D6105
      AND     M1310
      LD=     D2503 D6113
      AND=    D2504 D6114
      AND=    D2505 D6115
      AND     M1311
      ORB
      LD=     D2503 D6123
      AND=    D2504 D6124
      AND=    D2505 D6125
      AND     M1312
      ORB
      LD=     D2503 D6133
      AND=    D2504 D6134
      AND=    D2505 D6135
      AND     M1313
      ORB
      LD=     D2503 D6143
      AND=    D2504 D6144
      AND=    D2505 D6145
      AND     M1314
      ORB
      LD=     D2503 D6153
      AND=    D2504 D6154
      AND=    D2505 D6155
      AND     M1315
      ORB
      LD=     D2503 D6163
      AND=    D2504 D6164
      AND=    D2505 D6165
      AND     M1316
      ORB
      LD=     D2503 D6173
      AND=    D2504 D6174
      AND=    D2505 D6175
      AND     M1317
      ORB
      LD=     D2503 D6183
      AND=    D2504 D6184
      AND=    D2505 D6185
      AND     M1318
      ORB
      LD=     D2503 D6193
      AND=    D2504 D6194
      AND=    D2505 D6195
      AND     M1319
      ORB
      ANB
      OUT     M1381
